Fanuc KAREL source: ks00040.KL

-- PROVISIONAL review KL for V940-1; original PC SHA256 8cd57458139b42c71fd9b30e9d9d2c9c69d57f8b873b9e1db781e04890767ac0
-- Incomplete behavior may be omitted. Consult companion uncertainty JSON. Do not deploy.
PROGRAM KS00040
%NOLOCKGROUP
BEGIN
  -- V9_ZERO_TABLE_METADATA_HINT layout=0001; no indexed target words; source/name/runtime held
  -- UNRESOLVED_PC offsets 5-13; opcodes 3F,75
  -- UNRESOLVED_PC offsets 18-27; opcodes 3F,75
  -- UNRESOLVED_PC offsets 32-45; opcodes 22,1D,23
  -- UNRESOLVED_PC offsets 50-54; opcodes 7F
END KS00040
